IF poti_max_s16 <= 950 THEN
	poti_emax_s16 := poti_max_s16 + 50;
ELSE
	poti_emax_s16 := 1000;
END_IF

(* read jostick poti *)
poti_raw_s16 := inext_getPoti( PotiChannel_u32, poti_min_s16, poti_max_s16, poti_emin_s16, poti_emax_s16 );
poti_raw_s16 := LIMIT (0, poti_raw_s16, ST_RANGE);

poti_s16:=calc_deadband(poti_raw_s16, Deadband_s16);
END_FUNCTION_BLOCK

(* POU 10_Inputs/Function Blocks/in_joystick_fb, ST *)
FUNCTION_BLOCK in_joystick_fb
VAR_OUTPUT
	poti_s16			: INT;	(*	poti position, [-1000 .. 1000]	Unit = 0.1%*)
	poti_raw_s16	: INT;	(*	poti position without deadband *)
END_VAR
VAR
	poti_min_s16	: INT;
	poti_mid_s16	: INT;
	poti_max_s16	: INT;
	poti_emin_s16	: INT;
	poti_emax_s16	: INT;
END_VAR
VAR_INPUT
	PotiAdjust_s16	: INT;
	PotiMiddle_s16	: INT;
	Deadband_s16	: INT;
	PotiChannel_u32: DWORD;
END_VAR
(* get poti adjustment values *)
poti_min_s16 := inext_getPotiMin( PotiAdjust_s16 );
poti_max_s16 := inext_getPotiMax( PotiAdjust_s16 );
poti_mid_s16 := inext_getPotiMid( PotiMiddle_s16 );

(*derive error thresholds from adjustment values *)
IF poti_min_s16 >= 50 THEN
	poti_emin_s16 := poti_min_s16 - 50;
ELSE
	poti_emin_s16 := 0;
END_IF

IF poti_max_s16 <= 950 THEN
	poti_emax_s16 := poti_max_s16 + 50;
ELSE
	poti_emax_s16 := 1000;
END_IF
(* read jostick poti *)
poti_raw_s16 := inext_getPotiDir(	PotiChannel_u32,
												poti_min_s16,
												poti_max_s16,
												poti_mid_s16,
												poti_emin_s16,
												poti_emax_s16 );

poti_s16:=calc_deadband(poti_raw_s16, Deadband_s16);
END_FUNCTION_BLOCK

(* POU 05_Basic_Calc/isRegulationNow, ST *)
FUNCTION_BLOCK isRegulationNow
VAR_INPUT
	RAW_SIGNAL				: INT;				(* Непосредственно сигнал *)
	error						: INT;				(* Погрешность *)
	timer_regul				: TON;				(* Таймер для защиты от помех *)
	timer_reg_in			: BOOL;				(* Вход таймера *)
END_VAR
VAR_OUTPUT
	isRegulationNow		: BOOL;				(* Происходит ли регуливка в данный момент *)
END_VAR
VAR
	buffer					: INT := 0;			(* Буффер для хранения значения *)
	buffer_state			: INT;				(* Состояние буффера *)
END_VAR
VAR CONSTANT
	AMOUNT_OF_REG_CYCLES	: INT	:= 10;		(* Количество циклов, допускающее скачок *)
END_VAR
timer_regul(in:= timer_reg_in, PT:= INT_TO_TIME(CYCLE * AMOUNT_OF_REG_CYCLES), Q=> , ET=> );
	CASE buffer_state OF
		0:
			buffer			:=	RAW_SIGNAL;
			buffer_state	:=	1;
		1:
			IF ABS(buffer-RAW_SIGNAL) > error THEN
				timer_reg_in		:= TRUE;
				IF timer_regul.Q THEN
					isRegulationNow	:=	TRUE;
					buffer_state		:=	0;
					timer_reg_in		:= FALSE;
				END_IF
			ELSE
				isRegulationNow	:=	FALSE;
				timer_reg_in		:= FALSE;
			END_IF
	END_CASE
END_FUNCTION_BLOCK

(* POU 05_Basic_Calc/Lowpass_calc, ST *)
FUNCTION_BLOCK Lowpass_calc
VAR_INPUT
	iDivisor: INT;
	iInput: INT;
END_VAR
VAR_OUTPUT
	iOutput: INT;
END_VAR
VAR
	iY: DINT;
END_VAR
(*The calculation of the divisor ( iTime:constant / iCycle_time) is done in the initialization function block "Lowpass_init" *)

iY :=iY - (iY / iDivisor) + iInput;
iOutput := DINT_TO_INT(iY / iDivisor);
END_FUNCTION_BLOCK

(* POU 05_Basic_Calc/Lowpass_init, ST *)
FUNCTION_BLOCK Lowpass_init
VAR_INPUT
	tTime_constant: TIME;
	iCycle_time: INT;
END_VAR
VAR_OUTPUT
END_VAR
VAR_IN_OUT
	iDivisor: INT;
END_VAR

VAR
	iTime_constant:INT;
END_VAR
iTime_constant:=TIME_TO_INT(tTime_constant);

iCycle_time := MAX(1,iCycle_time );	(*not zero*)
iTime_constant := LIMIT(iCycle_time, iTime_constant, iTime_constant); (*Time constant min. Cycle_time*)

iDivisor:=iTime_constant / iCycle_time;
END_FUNCTION_BLOCK

(* POU 05_Basic_Calc/roundingTo5, ST *)
FUNCTION roundingTo5 : UINT 	(* Функция окргуляет число до ближайшего кратного (5 * order) числа *)
VAR_INPUT
	in_number_u16	: UINT;		(* Число, которое нужно округлить *)
	order				: UINT;		(* Порядок до которого округлять. 1 – до кратного 5ти, 10 – до кратного 50ти, и тд... *)
END_VAR
VAR
	div_part			: REAL;		(* Целое число *)
	aux_num			: UINT;		(* вспомогательная переменная для отслеживания округления до меньшего целого *)
	dec_part			: REAL;		(* десятая часть числа *)
END_VAR
VAR CONSTANT
	LOW_ROUND		: REAL := 0.25;
	HIGH_ROUND		: REAL := 0.75;
END_VAR
IF order < 1 THEN
	roundingTo5 := in_number_u16;
ELSE
	IF order < 10 THEN
		order := 1;
	ELSIF order < 100 THEN
		order := 10;
	ELSIF order < 1000 THEN
		order := 100;
	ELSIF order < 10000 THEN
		order := 1000;
	ELSE
		order := 10000;
	END_IF

	div_part	:= UINT_TO_REAL(in_number_u16) / (order * 10);
	aux_num	:= REAL_TO_UINT(div_part);
	
	IF UINT_TO_REAL(aux_num) > div_part THEN
		aux_num := aux_num - 1;
	END_IF

	dec_part	:= ABS(div_part - UINT_TO_REAL(aux_num));

	IF dec_part >= LOW_ROUND AND  dec_part < HIGH_ROUND THEN
		dec_part := 0.5;
	ELSIF dec_part < LOW_ROUND THEN
		dec_part := 0.0;
	ELSE
		dec_part := 1.0;
	END_IF

	roundingTo5 := (aux_num * (order * 10) + REAL_TO_UINT(dec_part * (order * 10)));
END_IF
END_FUNCTION

(* POU 05_Basic_Calc/eeprom_operations/saveValue_if_Changed, ST *)
FUNCTION saveValue_if_Changed : INT
(* Функция выполняет проверку параметра EEPROM.
	В случае, если параметр изменился, то производим сохранение в память EEPROM *)
VAR_INPUT
	isSave_enabled_b8		: BOOL;			(* Флаг - Внесение изменений в память EEPROM разрешено *)

	EEP_num					: INT;			(* Номер параметра в EEPROM*)
	param_s16				: INT;			(* Параметр, который нужно проверить и пересохранить *)
END_VAR
VAR
	ee_param_s16			: INT;			(* Значение параметра в памяти EEPROM *)

END_VAR
	IF isSave_enabled_b8 THEN

		(* Получение актуального значения параметра в EEPROM *)
		ee_param_s16 := ree_getValue(getEEP_Page(EEP_num), getEEP_Index(EEP_num));

		IF param_s16 <> ee_param_s16 THEN
		(* Если параметр не соответствует значению в EEPROM, то сохраняем измененный параметр в память EEPROM *)

			saveValue_if_Changed := ee_saveValue(getEEP_Page(EEP_num), getEEP_Index(EEP_num), param_s16);

		END_IF

	END_IF
END_FUNCTION

(* POU 05_Basic_Calc/set_poti_value, ST *)
FUNCTION set_poti_value : INT
(* Функция задания калибровочного значения потенциометра по его минимальному и максимальному значениям *)
(* Функция возвращает -1, если введены не верные входные параметры *)
VAR_INPUT
	in_min_mV_s16		: INT;		(* Минимальное значение потенциометра, мВ *)
	in_max_mV_s16		: INT;		(* Максимальное значение потенциометра, мВ *)
	U_lim_mV_s16		: INT;		(* Максимально допустимое напряжение на входе, мВ *)
END_VAR
VAR
	U_half_lim_s16		: INT;		(* Половина диапазона допустимого напряжения*)
	dig_min_raw_s16	: INT;		(* Сконвертированное минимальное значение потенциометра, [0; 255] *)
	dig_max_raw_s16	: INT;		(* Сконвертированное максимальное значение потенциометра, [256; 511] *)
	dig_min_s16			: WORD;		(* Сконвертированное мин. значение потенциометра *)
	dig_max_s16			: WORD;		(* Сконвертированное макс. значение потенциометра *)
END_VAR
	(* Получение границ диапазона для минимального и максимального значения потенциометра *)
	U_half_lim_s16 := U_lim_mV_s16 / 2;

		(* Проверка на правильность входных данных *)
	IF in_min_mV_s16 > U_half_lim_s16	OR
		in_max_mV_s16 < U_half_lim_s16	THEN

		(* Входные данные не верные *)
		set_poti_value := -1;
	ELSE
		(* Входные данные верные *)

		(* Конвертация значений потенциометра в цифровые значения *)
		dig_min_raw_s16 := conv_mV_to_dig(in_min_mV_s16, U_lim_mV_s16);
		dig_max_raw_s16 := conv_mV_to_dig(in_max_mV_s16, U_lim_mV_s16);

		(* Проверка выполнения конвертации *)
		IF dig_min_raw_s16 = -1 OR
			dig_max_raw_s16 = -1 THEN
			(* Конвертация не выполнена, входные данные не верные *)
			set_poti_value := -1;
		ELSE
			(* Конвертация выполнена *)

			(* Пересчет калибровочного значения *)
			dig_min_s16		:= SHL((INT_TO_WORD(dig_min_raw_s16) AND 16#00FF), 8);
			dig_max_s16		:= (INT_TO_WORD(511 - dig_max_raw_s16) AND 16#00FF);

			(* Получение готового калибровочного значения потенциометра *)
			set_poti_value	:= WORD_TO_INT(dig_min_s16 OR dig_max_s16);
		END_IF
	END_IF
END_FUNCTION

(* POU 30_Outputs/setProp, ST *)
FUNCTION setProp : UINT
VAR_INPUT
	Chn_u32		: UDINT;
	i_Input_s32	: DINT;
	Imin_s16		: INT;
	Imax_s16		: INT;
END_VAR
VAR
	i_mA_u16		: UINT;
END_VAR
(* Обратить внимание: если на вход i_Input_s32 подается 0, то минимальный ток игнорируется *)
IF i_Input_s32 > 0 AND i_Input_s32 <= ST_RANGE THEN
	i_mA_u16 := DINT_TO_UINT (  i_Input_s32 * ( Imax_s16 - Imin_s16) / ST_RANGE + Imin_s16 );
ELSE
	i_mA_u16 := 0;
END_IF

out(Chn_u32, i_mA_u16);
setProp := i_mA_u16;
END_FUNCTION

(* POU 05_Basic_Calc/tact_button, CFC *)
FUNCTION_BLOCK tact_button
VAR_INPUT
	button:	BOOL;
END_VAR
VAR_OUTPUT
	state:	BOOL;
END_VAR
VAR
	rtr1:	R_TRIG;
	rs1: 	RS;
END_VAR
VAR (* helpers for the ST form of the networks *)
	_t254 : BOOL;
	_t258 : BOOL;
END_VAR
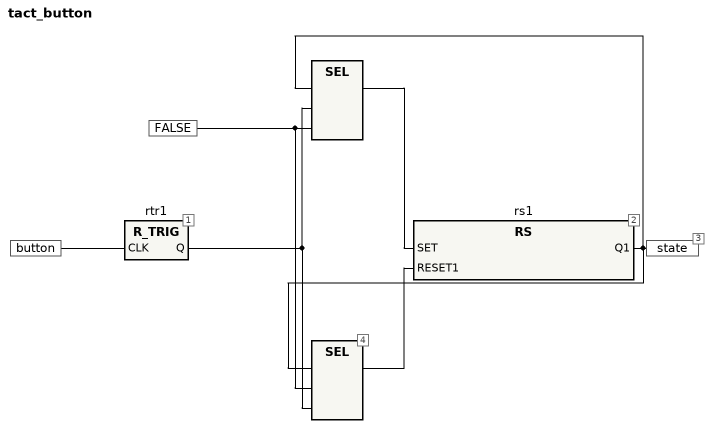
_CFC_ (* Continuous Function Chart, elements in execution order *)
#0 SEL(#2.Q1, #1.Q, FALSE)
#1 rtr1:R_TRIG(CLK: button)
#2 rs1:RS(SET: #0, RESET1: #4)
#3 state <= #2.Q1
#4 SEL(#2.Q1, FALSE, #1.Q)
_END_CFC_
(* the same logic as Structured Text *)
_t254 := SEL(rs1.Q1, rtr1.Q, FALSE);
rtr1(CLK := button);
rs1(SET := _t254, RESET1 := _t258);
state := rs1.Q1;
_t258 := SEL(rs1.Q1, FALSE, rtr1.Q);
END_FUNCTION_BLOCK
